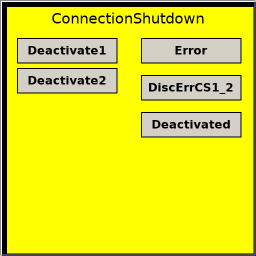
VISUALIZATION V_PH_CONNECTIONSHUTDOWN  // 256x256
VAR_INPUT
	stSafetyConnectionShutdown				:ST_SAFETY_FBCONNECTIONSHUTDOWN;
	
	
END_VAR
    Rectangle (2,2 256x256), colour toggle: stSafetyConnectionShutdown.bGeneralError
    Label (5,6 246x25), "ConnectionShutdown"
    RoundedRectangle (17,38 100x25), "Deactivate1", colour toggle: stSafetyConnectionShutdown.uStatus.stStatusWords.wInputs.8
    RoundedRectangle (17,68 100x25), "Deactivate2", colour toggle: stSafetyConnectionShutdown.uStatus.stStatusWords.wInputs.9
    RoundedRectangle (141,38 100x25), "Error", colour toggle: stSafetyConnectionShutdown.uStatus.stStatusWords.wOutputs.0
    RoundedRectangle (141,112 100x25), "Deactivated", colour toggle: stSafetyConnectionShutdown.uStatus.stStatusWords.wOutputs.1
    RoundedRectangle (141,75 100x25), "DiscErrCS1_2", colour toggle: stSafetyConnectionShutdown.uStatus.stStatusWords.wDiagnosis.0, invisible if: NOT stSafetyConnectionShutdown.uStatus.stStatusWords.wDiagnosis.0
    Textfield (17,226 234x25), text list: 'TL_FbStateCS', text index: stSafetyConnectionShutdown.eState
END_VISUALIZATION

(* stored: Version 1.1.0.1, ProductVersion 3.1.4024.4
   Visu V_PH_CONNECTIONSHUTDOWN: Id {82091db5-56ed-4d86-9771-dadfc97f6230} *)
